TYPE stAlarmHist :
STRUCT
	sDate:STRING(23);
	sTime:STRING(23);
	sMessage:STRING;
END_STRUCT
END_TYPE

(* stored: Version 1.1.0.1, ProductVersion 3.1.4024.11
   DUT stAlarmHist: Id {8812fa7d-3ca2-4850-b58b-5fba1ae93fd1} *)
